FUNCTION_BLOCK FB_SystemManager
VAR_INPUT
END_VAR
VAR_OUTPUT
END_VAR
VAR
	Devices : ARRAY [1..100] OF POINTER TO FB_Device;
	nRegisteredDevice :INT;
END_VAR

METHOD ExecuteDevices : BOOL
VAR
	idx: INT;
END_VAR
FOR idx :=1 TO nRegisteredDevice DO
	Devices[idx]^.Execute();
END_FOR
END_METHOD

METHOD FilterDeviceMacAddr : POINTER TO FB_Device;
VAR_INPUT
	macAdr: STRING;
END_VAR

VAR
	idx: INT;
END_VAR
FOR idx := 1 TO nRegisteredDevice DO
	IF Devices[idx]^.MacAddr = macAdr THEN
		FilterDeviceMacAddr := Devices[idx];
		RETURN;
	END_IF
END_FOR
END_METHOD

PROPERTY NumberOfRegisteredDevice : int
GET
END_GET
END_PROPERTY

METHOD registerDevice : BOOL
VAR_INPUT
	pDevice : REFERENCE TO FB_Device;
END_VAR
nRegisteredDevice := nRegisteredDevice + 1;
Devices[nRegisteredDevice] := ADR(pDevice);

ADSLOGSTR(msgCtrlMask := ADSLOG_MSGTYPE_ERROR, msgFmtStr := 'Registered Instance: %s', strArg := pDevice.Name);
END_METHOD

METHOD UnregisterDevice : BOOL
VAR_INPUT
END_VAR
END_METHOD

END_FUNCTION_BLOCK

(* stored: Version 1.1.0.1, ProductVersion 3.1.4024.9
   POU FB_SystemManager: Id {41ba94ab-514e-4adb-b068-8b35ea87ef43}, SpecialFunc None
   Method ExecuteDevices: Id {d1d33a3a-ca60-465f-8770-ad7b1efd40a6}
   Method FilterDeviceMacAddr: Id {9ebd669e-75d0-4aed-8a2e-b8e2bc1a84bc}
   Property NumberOfRegisteredDevice: Id {6b2cec84-de91-4179-98ea-1f915b3d7b80}
   Get Get: Id {1fb13df7-4ec2-4461-82a5-ea328342db46}
   Method registerDevice: Id {69150bb2-69da-4382-bcc6-522f37178f2b}
   Method UnregisterDevice: Id {270e34d5-79e4-4acc-9a41-054587a328b2} *)
